// TwinCAT 3 PLC project Inverse_Pendulum_PLC
// ProgramVersion: 3.1.4023.0
// libraries:
//   Tc2_Standard, * (Beckhoff Automation GmbH)
//   Tc2_System, * (Beckhoff Automation GmbH)
//   Tc3_Module, * (Beckhoff Automation GmbH)
//   Tc2_ControllerToolbox,3.4.3.0,Beckhoff Automation GmbH
// project tree:
//   DUTs/ E_RegulatorMode.TcDUT, ST_StateVariables.TcDUT
//   / PlcTask.TcTTO
//   POUs/ FB_InvertedPendulum.TcPOU, MAIN.TcPOU
// real-time tasks:
//   TASK PlcTask: cycle T#1ms, priority 20, ADS port 350

CONFIGURATION Inverse_Pendulum_PLC
    RESOURCE PLC ON TwinCAT3
        TASK PlcTask(INTERVAL := T#1ms, PRIORITY := 20);
        PROGRAM MAIN WITH PlcTask : MAIN;
    END_RESOURCE
END_CONFIGURATION

// ---- DUTs/E_RegulatorMode.TcDUT
{attribute 'qualified_only'}
{attribute 'strict'}
TYPE E_RegulatorMode :
(
	eDisabled,
	ePID,
	eCascade
);
END_TYPE

// ---- DUTs/ST_StateVariables.TcDUT
TYPE ST_StateVariables :
STRUCT
	fX : 	LREAL := 0.0;
	fXD : 	LREAL := 0.0;
	fTheta : LREAL := 0.0;
	fThetaD : LREAL := 0.0;
END_STRUCT
END_TYPE

// ---- POUs/MAIN.TcPOU
PROGRAM MAIN
VAR
	//HMI stuff
	bHMI_ForceStateVariables : BOOL := FALSE;
	stHMI_ForcedStateVariables : ST_StateVariables;
	fHMI_positionScale : LREAL; //scaling the displacement of the cart in HMI. There is probably a better way to do this.
	
	//Initialize simulator
	fInputForce : LREAL := 0.0;
	stStateVariables : ST_StateVariables;
	stInitialStateVariables : ST_StateVariables := (fX := 0.0, fXD := 0.0, fTheta := 0.000, fThetaD := 0.0);
	fbInvertedPendulum : FB_InvertedPendulum(
		fMassPendulum := 1.0, 
		fMassCart := 3.0, 
		fLengthPendulum := 0.5, 
		stInitialStateVariables := stInitialStateVariables,
		nCycleTimeMs:= 1);
		
	//Regulator
	fX_SP : LREAL := 0.0;
	fThetaSP : LREAL := 0.0;
	eRegulatorMode: E_RegulatorMode := E_RegulatorMode.eDisabled;
		
	//PID Controller for X (Outer loop)
	ePID_X_eMode : E_CTRL_MODE;
	stPID_X_settings : ST_CTRL_PID_PARAMS := (
		tCtrlCycleTime := T#10MS,
		tTaskCycleTime := T#1MS, 
		fKp := 0.2,  	 //P
		tTn := T#0MS,//I
		tTv := T#200MS,//D
		tTd := T#0MS,//Derivator filter
		fOutMaxLimit := 0.2,
		fOutMinLimit := -0.2,
		bPInTheFeedbackPath := FALSE,
		bDInTheFeedbackPath := FALSE,
		bARWOnIPartOnly := FALSE);
	fbPID_X : FB_CTRL_PID;
	
	//PID Controller for theta (Inner loop)
	ePID_Theta_eMode : E_CTRL_MODE;
	stPID_Theta_settings : ST_CTRL_PID_PARAMS := (
		tCtrlCycleTime := T#1MS, 
		tTaskCycleTime := T#1MS, 
		fKp := 200,  //P
		tTn := T#0MS,//I
		tTv := T#40MS,//D
		tTd := T#0MS,//Derivator filter
		fOutMaxLimit := 100,
		fOutMinLimit := -100,
		bPInTheFeedbackPath := FALSE,
		bDInTheFeedbackPath := FALSE,
		bARWOnIPartOnly := FALSE);
	fbPID_Theta : FB_CTRL_PID;
END_VAR

CASE eRegulatorMode OF
	E_RegulatorMode.eDisabled:
		ePID_X_eMode := E_CTRL_MODE.eCTRL_MODE_IDLE;
		ePID_Theta_eMode := E_CTRL_MODE.eCTRL_MODE_IDLE;
		
	E_RegulatorMode.ePID:
		ePID_X_eMode := E_CTRL_MODE.eCTRL_MODE_MANUAL;
		ePID_Theta_eMode := E_CTRL_MODE.eCTRL_MODE_ACTIVE;
			
	E_RegulatorMode.eCascade:
		ePID_X_eMode := E_CTRL_MODE.eCTRL_MODE_ACTIVE;
		ePID_Theta_eMode := E_CTRL_MODE.eCTRL_MODE_ACTIVE;
END_CASE

fbPID_X(
	fSetpointValue := fX_SP, 
	fActualValue := stStateVariables.fX,
	fManSyncValue := 0.0,
	eMode := ePID_X_eMode, 
	stParams := stPID_X_settings);
	fThetaSP := fbPID_X.fOut;

fbPID_Theta(
	fSetpointValue := fThetaSP, 
	fActualValue := stStateVariables.fTheta, 
	eMode := ePID_Theta_eMode, 
	stParams := stPID_Theta_settings);
	fInputForce := fbPID_Theta.fOut*-1;
	
stStateVariables := fbInvertedPendulum.Simulate(fForce := fInputForce);

IF bHMI_ForceStateVariables THEN
	fbInvertedPendulum.ForceStateVariables(stNewStateVariables := stHMI_ForcedStateVariables);
	bHMI_ForceStateVariables := FALSE;
END_IF

fHMI_positionScale := stStateVariables.fX * 200;

END_PROGRAM

// ---- POUs/FB_InvertedPendulum.TcPOU
FUNCTION_BLOCK FB_InvertedPendulum
VAR
	stStateVariables : ST_StateVariables;
	fXDD : LREAL;	//[m/s^2] Acceleratiomn of cart
	fThetaDD : LREAL;	//[rad/s^2] Angular acceleration Pendulum
	fMp : LREAL; 		//[kg] Mass of pendulum
	fMc : LREAL; 		//[kg] Mass of cart
	fL : LREAL;  		//[m] Length of pendulum
	fCycleTimeSeconds : LREAL;
END_VAR

VAR CONSTANT
	fG : LREAL := 9.81; //[m/s^2] Gravity
END_VAR

METHOD FB_init : BOOL
VAR_INPUT
	bInitRetains : BOOL; // if TRUE, the retain variables are initialized (warm start / cold start)
	bInCopyCode : BOOL;  // if TRUE, the instance afterwards gets moved into the copy code (online change)
	fMassPendulum : LREAL; 
	fMassCart : LREAL; 
	fLengthPendulum : LREAL; 
	stInitialStateVariables : ST_StateVariables;
	nCycleTimeMs : INT;
END_VAR
fMp := fMassPendulum;
fMc := fMassCart;
fL := fLengthPendulum;
fCycleTimeSeconds := nCycleTimeMs / 1000.0;
stStateVariables := stInitialStateVariables;
FB_Init := TRUE;
END_METHOD

METHOD PUBLIC ForceStateVariables
VAR_INPUT
	stNewStateVariables: ST_StateVariables;
END_VAR
stStateVariables := stNewStateVariables;
END_METHOD

METHOD PUBLIC Simulate : ST_StateVariables
VAR
	fCosTheta : LREAL;
	fSinTheta : LREAL;
END_VAR

VAR_INPUT
	fForce : LREAL; //[N]
END_VAR

VAR_OUTPUT
	stStateVariablesOutput : ST_StateVariables;
END_VAR
fCosTheta := COS(stStateVariables.fTheta);
fSinTheta := SIN(stStateVariables.fTheta);

fXDD := (fForce 
		+ fMp * fL * fSinTheta* stStateVariables.fThetaD * stStateVariables.fThetaD  
		- fMp * fG * fCosTheta * fSinTheta) 
		/(fMp + fMc - fMp * fCosTheta *fCosTheta);
		
fThetaDD := (fG * fSinTheta / fL)
			- (fForce * fCosTheta 
			+ fMp * fL * fSinTheta * fCosTheta * stStateVariables.fThetaD * stStateVariables.fThetaD
			- fMp * fG * fCosTheta*fCosTheta*fSinTheta)
			/ (fL * (fMp + fMc - fMp * fCosTheta * fCosTheta));

			
//Time integration
stStateVariables.fX := stStateVariables.fX + stStateVariables.fXD * fCycleTimeSeconds;
stStateVariables.fXD := stStateVariables.fXD + fXDD * fCycleTimeSeconds;

stStateVariables.fTheta := stStateVariables.fTheta + stStateVariables.fThetaD * fCycleTimeSeconds;
stStateVariables.fThetaD := stStateVariables.fThetaD + fThetaDD * fCycleTimeSeconds;

Simulate := stStateVariables;
END_METHOD

END_FUNCTION_BLOCK
